// TIA Portal project "Backup" (V17)

(* hardware
DEVICE "S7-1200 station_1"  S7-1200 Station
   slot 0: "Rack_0"  S7-1200 Rack  Rack  V1.0
   slot 1: "PLC_1"  CPU 1212C DC/DC/DC  6ES7 212-1AE40-0XB0  V4.5
*)

// ===== PLC "PLC_1"  CPU 1212C DC/DC/DC =====

VAR_GLOBAL   // PLC tag table "Default tag table"
   "Start NO" AT %I0.0 : Bool;
   "Stop NC" AT %I0.1 : Bool;
   "Cam bien xylanh 1" AT %I0.2 : Bool;
   "Cam bien xylanh 2" AT %I0.3 : Bool;
   "Bang tai" AT %Q0.0 : Bool;
   "Xylanh1" AT %Q0.1 : Bool;
   "Xylanh2" AT %Q0.2 : Bool;
   "Master On" AT %M0.0 : Bool;
   "San pham 1" AT %M0.1 : Bool;
   "San pham 2" AT %M0.2 : Bool;
   "San pham 3" AT %M0.3 : Bool;
   "Tag_1" AT %M0.4 : Bool;
   "Tag_2" AT %M0.5 : Bool;
   "Tag_3" AT %M0.6 : Bool;
   "Tag_4" AT %M0.7 : Bool;
END_VAR

DATA_BLOCK "DKPLC"   // DB1
{ S7_Optimized_Access := 'FALSE' }
VERSION : 0.1
   VAR
      Start1 : Bool;
      Stop1 : Bool;
   END_VAR
BEGIN
END_DATA_BLOCK

DATA_BLOCK "PythonData"   // DB2
{ S7_Optimized_Access := 'FALSE' }
VERSION : 0.1
   VAR
      "Gia tri QR" : Int;
   END_VAR
BEGIN
END_DATA_BLOCK

// folder: System blocks/Program resources

DATA_BLOCK "IEC_Timer_0_DB"   // DB3
{ S7_Optimized_Access := 'TRUE' }
AUTHOR : Simatic
FAMILY : IEC
NAME : IEC_TMR
VERSION : 1.0
// stored: InstanceOfName IEC_TIMER
"IEC_TIMER"
BEGIN
END_DATA_BLOCK

DATA_BLOCK "IEC_Timer_0_DB_1"   // DB4
{ S7_Optimized_Access := 'TRUE' }
AUTHOR : Simatic
FAMILY : IEC
NAME : IEC_TMR
VERSION : 1.0
// stored: InstanceOfName IEC_TIMER
"IEC_TIMER"
BEGIN
END_DATA_BLOCK

DATA_BLOCK "IEC_Timer_0_DB_2"   // DB5
{ S7_Optimized_Access := 'TRUE' }
AUTHOR : Simatic
FAMILY : IEC
NAME : IEC_TMR
VERSION : 1.0
// stored: InstanceOfName IEC_TIMER
"IEC_TIMER"
BEGIN
END_DATA_BLOCK

// folder: (top level)

ORGANIZATION_BLOCK "Main"   // OB1, LAD, ProgramCycle
TITLE = "Main Program Sweep (Cycle)"
{ S7_Optimized_Access := 'TRUE' }
VERSION : 0.1
   VAR_INPUT
      Initial_Call : Bool;   // Initial call of this OB
      Remanence : Bool;   // =True, if remanent data are available
   END_VAR
   VAR_TEMP   // added for the SCL form of the ladder/FBD networks
      _w1 : Bool;
      _w2 : Bool;
      _w3 : Bool;
      _w4 : Bool;
   END_VAR
BEGIN

REGION Network 1: đóng mở hệ thống
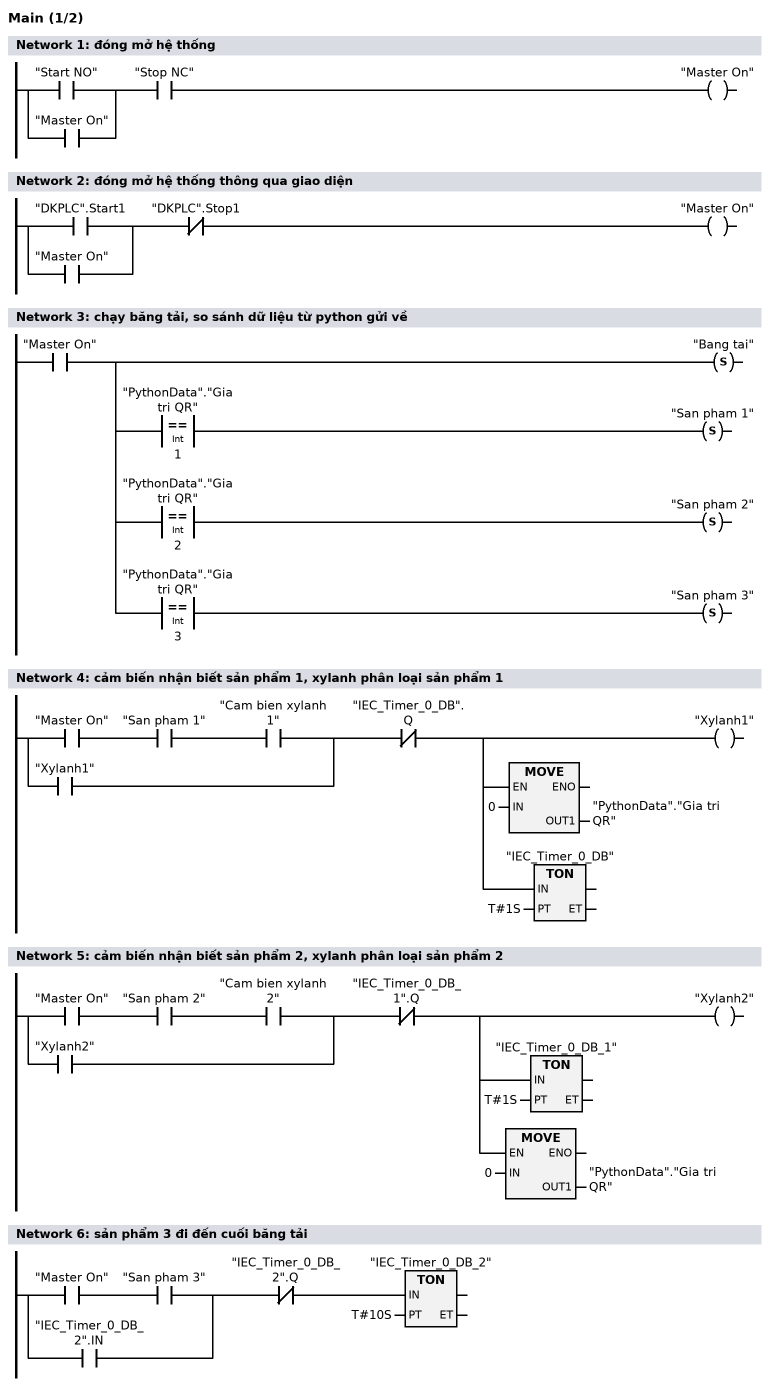
   RUNG wire#powerrail
      Contact( "Start NO" )
      wire#w1
      Contact( "Stop NC" )
      Coil( "Master On" )
   END_RUNG
   RUNG wire#powerrail
      Contact( "Master On" )
   END_RUNG wire#w1
   // the same network as SCL:
   "Master On" := ("Start NO" OR "Master On") AND "Stop NC";
END_REGION

REGION Network 2: đóng mở hệ thống thông qua giao diện
   RUNG wire#powerrail
      Contact( "DKPLC".Start1 )
      wire#w1
      I_Contact( "DKPLC".Stop1 )
      Coil( "Master On" )
   END_RUNG
   RUNG wire#powerrail
      Contact( "Master On" )
   END_RUNG wire#w1
   // the same network as SCL:
   "Master On" := ("DKPLC".Start1 OR "Master On") AND NOT "DKPLC".Stop1;
END_REGION

REGION Network 3: chạy băng tải, so sánh dữ liệu từ python gửi về
   RUNG wire#powerrail
      Contact( "Master On" )
      wire#w1
      S_Coil( "Bang tai" )
   END_RUNG
   RUNG wire#w1
      { S7_Templates := "SrcType := Int" } EQ_Contact(in1 := "PythonData"."Gia tri QR", in2 := 1)
      S_Coil( "San pham 1" )
   END_RUNG
   RUNG wire#w1
      { S7_Templates := "SrcType := Int" } EQ_Contact(in1 := "PythonData"."Gia tri QR", in2 := 2)
      S_Coil( "San pham 2" )
   END_RUNG
   RUNG wire#w1
      { S7_Templates := "SrcType := Int" } EQ_Contact(in1 := "PythonData"."Gia tri QR", in2 := 3)
      S_Coil( "San pham 3" )
   END_RUNG
   // the same network as SCL:
   IF "Master On" THEN "Bang tai" := TRUE; END_IF;
   IF "Master On" AND ("PythonData"."Gia tri QR" = 1) THEN "San pham 1" := TRUE; END_IF;
   IF "Master On" AND ("PythonData"."Gia tri QR" = 2) THEN "San pham 2" := TRUE; END_IF;
   IF "Master On" AND ("PythonData"."Gia tri QR" = 3) THEN "San pham 3" := TRUE; END_IF;
END_REGION

REGION Network 4: cảm biến nhận biết sản phẩm 1, xylanh phân loại sản phẩm 1
   "Xylanh1" := (("Master On" AND "San pham 1" AND "Cam bien xylanh 1") OR "Xylanh1") AND NOT "IEC_Timer_0_DB".Q;
   IF "Xylanh1" THEN "PythonData"."Gia tri QR" := 0; END_IF;
   "IEC_Timer_0_DB".TON(IN := "Xylanh1", PT := T#1S);
END_REGION

REGION Network 5: cảm biến nhận biết sản phẩm 2, xylanh phân loại sản phẩm 2
   "Xylanh2" := (("Master On" AND "San pham 2" AND "Cam bien xylanh 2") OR "Xylanh2") AND NOT "IEC_Timer_0_DB_1".Q;
   "IEC_Timer_0_DB_1".TON(IN := "Xylanh2", PT := T#1S);
   IF "Xylanh2" THEN "PythonData"."Gia tri QR" := 0; END_IF;
END_REGION

REGION Network 6: sản phẩm 3 đi đến cuối băng tải
   "IEC_Timer_0_DB_2".TON(IN := (("Master On" AND "San pham 3") OR "IEC_Timer_0_DB_2".IN) AND NOT "IEC_Timer_0_DB_2".Q,
                          PT := T#10S);
END_REGION

REGION Network 7: reset băng tải và các sản phẩm
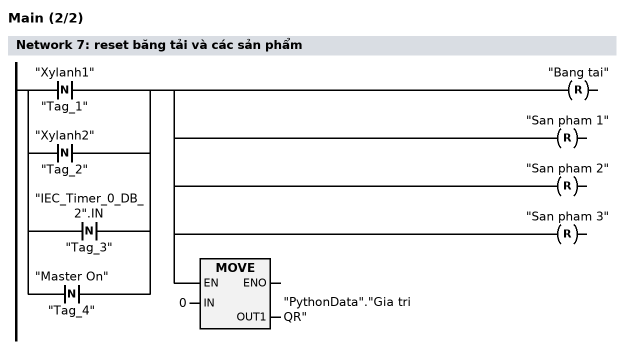
   RUNG wire#powerrail
      N_Contact(operand := "Xylanh1", bit := "Tag_1")
      wire#w1
      R_Coil( "Bang tai" )
   END_RUNG
   RUNG wire#powerrail
      N_Contact(operand := "Xylanh2", bit := "Tag_2")
   END_RUNG wire#w1
   RUNG wire#powerrail
      N_Contact(operand := "IEC_Timer_0_DB_2".IN, bit := "Tag_3")
   END_RUNG wire#w1
   RUNG wire#powerrail
      N_Contact(operand := "Master On", bit := "Tag_4")
   END_RUNG wire#w1
   RUNG wire#w1
      R_Coil( "San pham 1" )
   END_RUNG
   RUNG wire#w1
      R_Coil( "San pham 2" )
   END_RUNG
   RUNG wire#w1
      R_Coil( "San pham 3" )
   END_RUNG
   RUNG wire#w1
      Move(in := 0, out1 => "PythonData"."Gia tri QR")
   END_RUNG
   // the same network as SCL:
   #_w1 := NOT "Xylanh1" AND "Tag_1";   // falling edge of "Xylanh1"
   "Tag_1" := "Xylanh1";
   #_w2 := NOT "Xylanh2" AND "Tag_2";   // falling edge of "Xylanh2"
   "Tag_2" := "Xylanh2";
   #_w3 := NOT "IEC_Timer_0_DB_2".IN AND "Tag_3";   // falling edge of "IEC_Timer_0_DB_2".IN
   "Tag_3" := "IEC_Timer_0_DB_2".IN;
   #_w4 := NOT "Master On" AND "Tag_4";   // falling edge of "Master On"
   "Tag_4" := "Master On";
   IF #_w1 OR #_w2 OR #_w3 OR #_w4 THEN
       "Bang tai" := FALSE;
       "San pham 1" := FALSE;
       "San pham 2" := FALSE;
       "San pham 3" := FALSE;
       "PythonData"."Gia tri QR" := 0;
   END_IF;
END_REGION
END_ORGANIZATION_BLOCK